{attribute 'GeneratedUsingTerminal: EP2328-1061-0016'}
{attribute addProperty BoxType "EP2328-1061-0016"}
{attribute addProperty Id "OutputAT %Q*BOOL1"}
{attribute addProperty CRC "1120571895"}
{attribute addProperty Size "1"}
TYPE DO_X04_Pin4_Output_42CA91F7 :
STRUCT
	{attribute addProperty Name "Output"}
	Output AT %Q* : BOOL;
END_STRUCT
END_TYPE

(* stored: Version 1.2.0.0, ProductVersion 3.1.4024.9
   DUT DO_X04_Pin4_Output_42CA91F7: Id {d14be715-9c67-4841-85cf-1f8506e4471e} *)
